FUNCTION_BLOCK SubRoutineAutoMode EXTENDS TcoCore.TcoSequencer
VAR
    _counter : int :=1 ;
END_VAR

_counter := _counter + 1;

(*~
	<docu>
		<summary>
			Main method of the sequener. Custom code needs to be placed here. The sequencer is executed by call of InstanceName.Run() method.
			This method is abstract, and it must be overridden in derived block.
		</summary>
	</docu>
~*)
METHOD PROTECTED Main : BOOL
VAR_INST
    simTime : INT := 150;
END_VAR
IF (step(100, TRUE, 'SubRoutine Schritt eins, geht los')) THEN

    StepCompleteWhen(station.counter2 MOD simTime = 0);

END_IF

IF (step(200, TRUE, 'Sub ROutine Schritt 2')) THEN
    StepCompleteWhen(station.counter2 MOD simTime = 0);
END_IF

IF (step(300, TRUE, ' SubRoutine Schritt 3,')) THEN
    StepCompleteWhen(station.counter2 MOD simTime = 0);
END_IF

IF (step(400, TRUE, ' SubRoutine Schritt 4, wird beendet')) THEN
    ;
END_IF
END_METHOD

(*~
	<docu>
		<summary>
			This method is executed upon step completion.
			This method can be overridden in derived block by custom logic.
		</summary>			
	</docu>	
~*)
METHOD PROTECTED OnStepCompleted
station.counter2 := 1;
END_METHOD

PROPERTY Station : REFERENCE TO Test_Station
GET
VAR
    _station : POINTER TO Test_Station;
END_VAR
IF __QUERYPOINTER(_Parent,_station) THEN // Check if _Parent is Station001
	Station REF= _station^;              // If the check is successful dereference a pointer. simlar to THIS^ or SUPER^
END_IF
END_GET
END_PROPERTY

END_FUNCTION_BLOCK

(* stored: Version 1.1.0.1, ProductVersion 3.1.4024.9
   POU SubRoutineAutoMode: Id {0058c801-928e-0439-26d6-184635d0f0ae}, SpecialFunc None
   Method Main: Id {5b2f8d06-1073-0ba4-0dcc-aceba1450791}
   Method OnStepCompleted: Id {0e5655de-6ed3-0060-22cd-3a44463f146c}
   Property Station: Id {5420f3c0-2fcd-0571-3615-bc1c87107c55}
   Get Get: Id {5d74beaa-3167-0ec2-2db6-c089758b3fa6} *)
